// TIA Portal V20 export
TYPE "LER_FlexNet_Data"
// stored: Access Published
   STRUCT
      PUN : String[20];
      GM_PartNumber : String[8];
      OptionalData : String[12];
      TrackingID1 : String[32];   // Component 1 of the parent
      TrackingID1Attribute : String[20];   // Component 1 Attribute of the parent
      TrackingID2 : String[32];   // Component 2 of the parent
      TrackingID2Attribute : String[20];   // Component 2 Attribute of the parent
      TrackingID3 : String[32];   // Component 3 of the parent
      TrackingID3Attribute : String[20];   // Component 3 Attribute of the parent
      TrackingID4 : String[32];   // Component 4 of the parent
      TrackingID4Attribute : String[20];   // Component 4 Attribute of the parent
      TrackingID5 : String[32];   // Component 5 of the parent
      TrackingID5Attribute : String[20];   // Component 5 Attribute of the parent
      TrackingID6 : String[32];   // Component 6 of the parent
      TrackingID6Attribute : String[20];   // Component 6 Attribute of the parent
      TrackingID7 : String[32];   // Component 7 of the parent
      TrackingID7Attribute : String[20];   // Component 7 Attribute of the parent
      TrackingID8 : String[32];   // Component 8 of the parent
      TrackingID8Attribute : String[20];   // Component 8 Attribute of the parent
      TrackingID9 : String[32];   // Component 9 of the parent
      TrackingID9Attribute : String[20];   // Component 9 Attribute of the parent
      TrackingID10 : String[32];   // Component 10 of the parent
      TrackingID10Attribute : String[20];   // Component 10 Attribute of the parent
      PassFailFlagsByte : Char;
      Genealogy_Cnt : Byte;
      TransactionType : Byte;
      DataReady : Bool;
      Bypassed_Fault : Bool;
      DataReceivedByHost : Bool;
      ParentPartIsGood : Bool;
      ParentPartOnHold : Bool;
      TrackingComponent_1_IsGood : Bool;
      TrackingComponent_1_OnHold : Bool;
      TrackingComponent_2_IsGood : Bool;
      TrackingComponent_2_OnHold : Bool;
      TrackingComponent_3_IsGood : Bool;
      TrackingComponent_3_OnHold : Bool;
      TrackingComponent_4_IsGood : Bool;
      TrackingComponent_4_OnHold : Bool;
      TrackingComponent_5_IsGood : Bool;
      TrackingComponent_5_OnHold : Bool;
      TrackingComponent_6_IsGood : Bool;
      TrackingComponent_6_OnHold : Bool;
      TrackingComponent_7_IsGood : Bool;
      TrackingComponent_7_OnHold : Bool;
      TrackingComponent_8_IsGood : Bool;
      TrackingComponent_8_OnHold : Bool;
      TrackingComponent_9_IsGood : Bool;
      TrackingComponent_9_OnHold : Bool;
      TrackingComponent_10_IsGood : Bool;
      TrackingComponent_10_OnHold : Bool;
      White_LT_Solid : Bool;
      White_LT_Flash : Bool;
      Green_LT_Solid : Bool;
      Buzzer_Output : Bool;
      TimeStampYear : UInt;
      TimeStampMonth : USInt;
      TimeStampDate : USInt;
      TimeStampHour : USInt;
      TimeStampMinute : USInt;
      TimeStampSecond : USInt;
      Major_Spec_Version : Array[1..4] of Char;
      Minor_Spec_Version : Array[1..4] of Char;
      AOI_Revision : Int;
      PartPass : Bool;
      PartFail : Bool;
      DataReset : Bool;
      DryCycle : Bool;
      HQ_NOK : Bool;
      HQ_OK : Bool;
      ReTrigger_DataReady : Bool;
   END_STRUCT;
END_TYPE
